(*
	Function for motion control of single axis.
	Provides an interface to PLC Open motion control blocks.
	Controls linking of limit switches from slave to master axes.
*)
FUNCTION_BLOCK FB_AxisDrive
VAR_INPUT
END_VAR
VAR_IN_OUT
	AxisController		:	ST_AxisControl;
END_VAR
VAR_OUTPUT
END_VAR
VAR
	eCommandLatched		:	eMcCommand;		//Internally latched command signal, new commands cannot be issued until existing commands have completed.
	doneLatch	:	SR;						//Used to set done signal in AxisController DUT
	bDone		:	BOOL;					//Interal done flag which will be used for latching on an external done located in AxisController DUT
	iParam		:	INT:=1;					//index of NC parameters FBs, no 0 index on array so initialised to 1
	iIndex		:	UINT;					//index value used for limit coupling
	iMasterIndex		:	UINT;			//index value used for limit coupling
	
	//Boolean to store EnableFw and EnableBw of MCPower FB
	FwLimitsEnabled	:	BOOL;	
	BWLimitsEnabled	:	BOOL;
	
	mcDirection	:	MC_Direction;			//Direction control required in function blocks

(*
Motion Function blocks taken from the PLC OPEN standard as defined by PLC Open Standard
Function blocks commented out are yet to be added but the intention is to add these.
Those listed as //NOT IMPLEMENTED have come from the standard but Beckhoff do not support, 
these have been added just as a placeholder for future support.
*)
	//Not Implemented
	//MCReadDigitalInput		:	MC_ReadDigitalInput;			//NOT IMPLEMENTED		
	//MCReadDigitalOutput		:	MC_ReadDigitalOutput;			//NOT IMPLEMENTED	
	//MCWriteDigitalOutput		:	MC_WriteDigitalOutput;			//NOT IMPLEMENTED
	//MCReadActualTorque		:	MC_ReadActualTorque;			//NOT IMPLEMENTED	
	//MCReadAxisInfo			:	MC_ReadAxisInfo;				//NOT IMPLEMENTED	
	//MCReadMotionState			:	MC_ReadMotionState;				//NOT IMPLEMENTED
	//MCDigitalCamSwitch		:	MC_DigitalCamSwitch;			//NOT IMPLEMENTED
	//MCTorqueControl			:	MC_TorqueControl;				//NOT IMPLEMENTED		
	//MCPositionProfile			:	MC_PositionProfile;				//NOT IMPLEMENTED		
	//MCVelocityProfile			:	MC_VelocityProfile;				//NOT IMPLEMENTED		
	//MCAccelerationProfile		:	MC_AccelerationProfile;			//NOT IMPLEMENTED
	
	
	(* Administrative Function Blocks *)                                                                     
	MCReset						:	MC_Reset;											
	MCPower						:	MC_Power;										
	//MCReadStatus				:	MC_ReadStatus;					//Same as Axis.ReadStatus();						
	//MCReadAxisError			:	MC_ReadAxisError;									
	MCReadParameter				:	MC_ReadParameter;														
	MCWriteParameter			:	MC_WriteParameter;										
	MCWriteBoolParameter		:	MC_WriteBoolParameter;								
		
	//MCReadActualPosition		:	MC_ReadActualPosition;								
	//MCReadActualVelocity		:	MC_ReadActualVelocity;								
		
	MCSetPosition				:	MC_SetPosition;										
	//MCSetOverride				:	MC_SetOverride;										
	//MCTouchProbe				:	MC_TouchProbe;										
		
	//MCAbortTrigger			:	MC_AbortTrigger;									
	//MCAbortSuperposition		:	MC_AbortSuperposition;			//Listed as HaltSuperimposed in PLC Open standard	
	//MCCamTableSelect			:	MC_CamTableSelect;									
	
	(* Motion Function Blocks *)
	//MCHome					:	MC_Home;											
	MCJog						:	MC_Jog;												
	MCStop						:	MC_Stop;											
	//MCHalt					:	MC_Halt;											
	MCMoveAbsolute				:	MC_MoveAbsolute;									
	MCMoveRelative				:	MC_MoveRelative;									
	//MCMoveAdditive			:	MC_MoveAdditive;									
	//MCMoveSuperimposed		:	MC_MoveSuperimposed;								
	MCMoveVelocity				:	MC_MoveVelocity;									
	//MCMoveContinuousAbsolute	:	MC_MoveContinuousAbsolute;						
	//MCMoveContinuousRelative	:	MC_MoveContinuousRelative;						
	//MCMoveModulo				:	MC_MoveModulo;										
	
	(* Synchronised Motion Function Blocks *)		
	MCGearIn					:	MC_GearIn;											
	//MCGearInDyn				:	MC_GearInDyn;										
	MCGearInMultiMaster			:	MC_GearInMultiMaster;								
	MCGearOut					:	MC_GearOut;												                                                                                    
	//MCHaltPhasing				:	MC_HaltPhasing;										
	//MCPhasingAbsolute			:	MC_PhasingAbsolute;									
	//MCPhasingRelative			:	MC_PhasingRelative;										                                                                                                                                                 
	//MCCamIn					:	MC_CamIn;											
	//MCCamOut					:	MC_CamOut;											
	//MCCamScaling				:	MC_CamScaling;										                                                      
	//MCCamAdd					:	MC_CamAdd;											
	//MCCamExchange				:	MC_CamExchange;										
	//MCCamInV2					:	MC_CamIn_V2;		//REQUIRED FOR MULTICAMMING 	
	//MCCamRemove				:	MC_CamRemove;										
	//MCCamScalingV2			:	MC_CamScaling_V2;									

	(* Advanced Homing Steps and Finishing Moves *)
	MCFinishHoming			:	MC_FinishHoming;
	//MCHomeDirect			:	MC_HomeDirect;
	//MCAbortHoming			:	MC_AbortHoming;
	MCStepAbsoluteSwitch	:	MC_StepAbsoluteSwitch;
	//MCStepBlock			:	MC_StepBlock;
	//MCStepBlockLagBased	:	MC_StepBlockLagBased;
	//MCStepLimitSwitch		:	MC_StepLimitSwitch;
	//MCStepReferencePulse	:	MC_StepReferencePulse;
	
	
	(* Additional variable structures required for Advanced Homing *)
	//MCSignalRef			:	MC_Ref_Signal_Ref;
	StOptions				:	ST_Home_Options;
	StOptions2				:	ST_Home_Options2;
	StOptions3				:	ST_Home_Options3;
	StOptions4				:	ST_Home_Options4;
	MCHomingParameter		:	MC_HomingParameter;		//Must be passed between homing steps.		
							
		
END_VAR

AxisController.Axis.ReadStatus();
AxisController.fActPosition:= AxisController.Axis.NcToPlc.ActPos;
AxisController.fActVelocity:= AxisController.Axis.NcToPlc.ActVelo;
AxisController.bNegativeDirection:= AxisController.Axis.status.NegativeDirection;
AxisController.bPositiveDirection:= AxisController.Axis.Status.PositiveDirection;
AxisController.bCalibrated:= AxisController.Axis.Status.Homed;

//////////////////////////////////////////////////////////////////////
//     _   __  _____ ____    ____ _____  _  _____ _____ ____  		//
//    / \  \ \/ |_ _/ ___|  / ___|_   _|/ \|_   _| ____/ ___| 		//
//   / _ \  \  / | |\___ \  \___ \ | | / _ \ | | |  _| \___ \ 		//
//  / ___ \ /  \ | | ___) |  ___) || |/ ___ \| | | |___ ___) |		//
// /_/   \_/_/\_|___|____/  |____/ |_/_/   \_|_| |_____|____/ 		//
// 																	//
//////////////////////////////////////////////////////////////////////
                                                            
//Numerical representation for axis states - may use later for buffering functions.
IF AxisController.AXIS.Status.Disabled THEN
	AxisController.iAxisState:=		100;
ELSIF AxisController.AXIS.Status.StandStill THEN
	AxisController.iAxisState:=		200;
ELSIF AxisController.AXIS.Status.Homing	THEN
	AxisController.iAxisState:= 	300;
ELSIF AxisController.AXIS.Status.DiscreteMotion	THEN
	AxisController.iAxisState:=		400;
ELSIF AxisController.AXIS.Status.SynchronizedMotion	THEN
	AxisController.iAxisState:=		500;
ELSIF AxisController.AXIS.Status.ContinuousMotion	THEN
	AxisController.iAxisState:=		600;
ELSIF AxisController.AXIS.Status.Stopping	THEN
	AxisController.iAxisState:= 	700;	
ELSIF AxisController.AXIS.Status.Error THEN
	AxisController.iAxisState:=		999;	
ELSE
	AxisController.iAxisState:=		0;
END_IF

//////////////////////////////////////////////////////////////////////////////////////////
//  _     ___ __  __ ___ _____   ______        _____ _____ ____ _   _ _____ ____  		//
// | |   |_ _|  \/  |_ _|_   _| / ___\ \      / |_ _|_   _/ ___| | | | ____/ ___| 		//
// | |    | || |\/| || |  | |   \___ \\ \ /\ / / | |  | || |   | |_| |  _| \___ \ 		//
// | |___ | || |  | || |  | |    ___) |\ V  V /  | |  | || |___|  _  | |___ ___) |		//
// |_____|___|_|  |_|___| |_|   |____/  \_/\_/  |___| |_| \____|_| |_|_____|____/		//
//																						//
//////////////////////////////////////////////////////////////////////////////////////////

//Initialise Foward and Backward limits to the hardware limit switches for this axis
FwLimitsEnabled :=Limits.FwLimit[GVL.iAxis];
BwLimitsEnabled :=Limits.BwLimit[GVL.iAxis];

(*
Cycle through Limits.coupledFwLimit and Limits.coupledBwLimit.
Looking to see if any axes have the current axis (GVL.iAxis) listed as a master.
If this axis is listed as a master, check the hardware limits of that slave.
Gear ratio determines whether we are looking for a Forward or a Backward limit on the slave axis. 
If the limit switch is disabled, disable motion for this axis.
*)
FOR iIndex:=1 TO GVL.axisNumMax DO
	FOR iMasterIndex:=1 TO 5 DO
		//If listed as a master
		IF Limits.coupledFwLimit[iIndex][iMasterIndex].iMasterAxis = GVL.iAxis THEN
			//If forward limit linked to forward of slave, check forward limit of slave
			IF Limits.coupledFwLimit[iIndex][iMasterIndex].eLimitType=eLimitCoupling.FwSw AND NOT Limits.FwLimit[iIndex] THEN
				FwLimitsEnabled:=FALSE;
			END_IF
			//If forward limit linked to backwardof slave, check forward limit of slave
			IF Limits.coupledFwLimit[iIndex][iMasterIndex].eLimitType=eLimitCoupling.BwSw AND NOT Limits.BwLimit[iIndex] THEN
				FwLimitsEnabled:=FALSE;
			END_IF
			//If backward limit linked to forward of slave, check forward limit of slave
			IF Limits.coupledBwLimit[iIndex][iMasterIndex].eLimitType=eLimitCoupling.FwSw AND NOT Limits.FwLimit[iIndex] THEN
				BwLimitsEnabled:=FALSE;
			END_IF
			//If backward limit linked to backward of slave, check backward limit of slave
			IF Limits.coupledBwLimit[iIndex][iMasterIndex].eLimitType=eLimitCoupling.BwSw AND NOT Limits.BwLimit[iIndex] THEN
				BwLimitsEnabled:=FALSE;
			END_IF
		END_IF
	END_FOR
END_FOR

AxisController.bFwEnabled:=FwLimitsEnabled;		//Feedback to ST_AxisControl that forward positioning is available
AxisController.bBwEnabled:=BwLimitsEnabled;		//Feedback to ST_AxisControl that backward positioning is available

//////////////////////////////////////////////////////////
//  ____   _____        _______ ____    _   _ ____  	//
// |  _ \ / _ \ \      / | ____|  _ \  | | | |  _ \ 	//
// | |_) | | | \ \ /\ / /|  _| | |_) | | | | | |_) |	//
// |  __/| |_| |\ V  V / | |___|  _ <  | |_| |  __/ 	//
// |_|    \___/  \_/\_/  |_____|_| \_\  \___/|_|   		//
//														//
//////////////////////////////////////////////////////////
(*
Power up the axis.
Externally fed variables are bEnabled and fOverride, limits all controlled internally.
*)                                           
MCPower(
	Axis:=AxisController.Axis,
	Enable:=AxisController.bEnable,
	Enable_Positive:=FwLimitsEnabled,
	Enable_Negative:=BwLimitsEnabled,
	Override:=AxisController.fOverride,
	Status=>,
	Busy=>, 
	Active=>AxisController.bAxisReady,	//Maybe want a bPowered or bEnabled flag instead?
	Error=>,
	ErrorID=>
);

//////////////////////////////////////////////////////////////////////////////////////////////////////////
//  ____  _____    _    ____    ____   _    ____     _    __  __ _____ _____ _____ ____  ____  			//
// |  _ \| ____|  / \  |  _ \  |  _ \ / \  |  _ \   / \  |  \/  | ____|_   _| ____|  _ \/ ___| 			//
// | |_) |  _|   / _ \ | | | | | |_) / _ \ | |_) | / _ \ | |\/| |  _|   | | |  _| | |_) \___ \ 			//
// |  _ <| |___ / ___ \| |_| | |  __/ ___ \|  _ < / ___ \| |  | | |___  | | | |___|  _ < ___) |			//
// |_| \_|_____/_/   \_|____/  |_| /_/   \_|_| \_/_/   \_|_|  |_|_____| |_| |_____|_| \_|____/ 			//
//                                                                                           			//
//////////////////////////////////////////////////////////////////////////////////////////////////////////
(*
Check NC parameters available from MCReadParameter FB (17 in total)
See eRWParameter DUT for complete list or PLC OPEN documentation
To call all 17 from a single functionblock instance only 1 can be checked per cycle so there will be at minimum a 34 cycle delay checking each parameter
The MCReadParameter does also cover the functionality of MCReadBoolParameter so these booleans are separately converted from the MCReadParameter call
*)
MCReadParameter(Axis:=AxisController.AXIS,ParameterNumber:=iParam);
IF MCReadParameter.Valid THEN
	MCReadParameter.Enable:=FALSE;
	AxisController.fParameters[iParam]:=MCReadParameter.Value;
	iParam:= iParam+1;
	IF iParam>17 THEN
		iParam:=1;
	END_IF
ELSE
	MCReadParameter.Enable:=TRUE;
END_IF

//Convert LREALS to BOOLS


IF AxisController.fParameters[eRWParameter.EnableLimitPos]=1 THEN
	AxisController.bSoftLimPosEn:=TRUE;
ELSE
	AxisController.bSoftLimPosEn:=FALSE;
END_IF
IF AxisController.fParameters[eRWParameter.EnableLimitNeg]=1 THEN
	AxisController.bSoftLimNegEn:=TRUE;
ELSE
	AxisController.bSoftLimNegEn:=FALSE;
END_IF
IF AxisController.fParameters[eRWParameter.EnablePosLagMonitoring]=1 THEN
	AxisController.bPosLagEn:=TRUE;
ELSE
	AxisController.bPosLagEn:=FALSE;
END_IF

//////////////////////////////////////////////////////////////////////////////////////////////////////////
//  __  __  ____   _____ _   _ _   _  ____ _____ ___ ___  _   _    ____    _    _     _     ____  		//
// |  \/  |/ ___| |  ___| | | | \ | |/ ___|_   _|_ _/ _ \| \ | |  / ___|  / \  | |   | |   / ___| 		//
// | |\/| | |     | |_  | | | |  \| | |     | |  | | | | |  \| | | |     / _ \ | |   | |   \___ \ 		//
// | |  | | |___  |  _| | |_| | |\  | |___  | |  | | |_| | |\  | | |___ / ___ \| |___| |___ ___) |		//
// |_|  |_|\____| |_|    \___/|_| \_|\____| |_| |___\___/|_| \_|  \____/_/   \_|_____|_____|____/ 		//
//                                         																//                                                      
//////////////////////////////////////////////////////////////////////////////////////////////////////////
(*
Call MC Function Blocks and clear execute signals
Any MC function blocks added to the state machine must be called here with the given format.
Some FBs have slightly differing structures so these should aim to conform to the existing structure
Function blocks will hold done and error signals for 1 cycle with no execute held
*)
MCReadParameter(Axis:=AxisController.Axis);	//Reading in motion parameters, using one functionblock for all params means need to disable

MCReset(Axis:=AxisController.Axis);
MCReset.Execute:=FALSE;

MCWriteParameter(Axis:=AxisController.Axis);
MCWriteParameter.Execute:=FALSE;

MCWriteBoolParameter(Axis:=AxisController.Axis);
MCWriteBoolParameter.Execute:=FALSE;

MCSetPosition(Axis:=AxisController.Axis);
MCSetPosition.Execute:=FALSE;

MCMoveAbsolute(Axis:=AxisController.Axis);
MCMoveAbsolute.Execute:=FALSE;

MCMoveRelative(Axis:=AxisController.Axis);
MCMoveRelative.Execute:=FALSE;

MCGearIn(Slave:=AxisController.Axis, Master:=GVL.axes[AxisController.masterAxis].Axis);
MCGearIn.Execute:=FALSE;

MCGearInMultiMaster(Master1:=GVL.axes[AxisController.masterAxes[1].i].Axis,Master2:=GVL.axes[AxisController.masterAxes[2].i].Axis,Master3:=GVL.axes[AxisController.masterAxes[3].i].Axis,Master4:=GVL.axes[AxisController.masterAxes[4].i].Axis,Slave:=AxisController.Axis);
MCGearInMultiMaster.Enable:=FALSE;	//NOT EXECUTE AS FB ALLOWS CONTINUAL UPDATING OF RATIOS WHILST ENABLED

MCGearOut(Slave:=AxisController.Axis);
MCGearOut.Execute:=FALSE;

MCJog(Axis:=AxisController.Axis);
MCJog.JogBackwards:=FALSE;
MCJog.JogForward:=FALSE;

MCStepAbsoluteSwitch(Axis:=AxisController.Axis,Parameter:=MCHomingParameter);
MCStepAbsoluteSwitch.Execute:=FALSE;


MCFinishHoming(Axis:=AxisController.Axis,Parameter:=MCHomingParameter);
MCFinishHoming.Execute:=FALSE;

MCMoveVelocity(Axis:=AxisController.Axis);
MCMoveVelocity.Execute:=FALSE;

MCStop(Axis:=AxisController.Axis);
MCStop.Execute:=FALSE;

//////////////////////////////////////////////////////////////////////////////////////////////////////////////////////////////////////////////
//   ____ ___  __  __ __  __    _    _   _ ____     ____    _    ____  _____   ____ _____  _  _____ _____ __  __ _____ _   _ _____ ____ 	// 
//  / ___/ _ \|  \/  |  \/  |  / \  | \ | |  _ \   / ___|  / \  / ___|| ____| / ___|_   _|/ \|_   _| ____|  \/  | ____| \ | |_   _/ ___| 	//
// | |  | | | | |\/| | |\/| | / _ \ |  \| | | | | | |     / _ \ \___ \|  _|   \___ \ | | / _ \ | | |  _| | |\/| |  _| |  \| | | | \___ \ 	//
// | |__| |_| | |  | | |  | |/ ___ \| |\  | |_| | | |___ / ___ \ ___) | |___   ___) || |/ ___ \| | | |___| |  | | |___| |\  | | |  ___) |	//
//  \____\___/|_|  |_|_|  |_/_/   \_|_| \_|____/   \____/_/   \_|____/|_____| |____/ |_/_/   \_|_| |_____|_|  |_|_____|_| \_| |_| |____/	//
//																																			//
//////////////////////////////////////////////////////////////////////////////////////////////////////////////////////////////////////////////

(*
Internal statemachine to handle motion control flow and logic.
Functions are NOT called in this statemachine, these just update values given to the state machine. This was the method recommended by Beckhoff
The following basic wrapper should be used for adding new function blocks. Any that do not conform to this should be modified to conform
Notably some FBs have no .Done but do have .Active
	
	mcFunctionBlock.Execute		:=AxisController.bExecute;
	mcFunctionBlock.misc1..n	:=AxisController.misc1..n;
	
	bDone:=mcFunctionBlock.Done;
	AxisController.bBusy:= mcFunctionBlock.Busy;
	
	If mcFunctionBlock.Error THEN
		AxisController.bError:=TRUE;
		AxisController.iErrorID:= mcFunctionBlock.ErrorID;
	END_IF
	IF NOT mcFunctionBlock.Busy THEN
		eCommandLatched:=eMcCommand.Idle;
	END_IF
	
Function block specific parameters should be added to the ST_AxisControl if not already listed
eCommandLatched is currently being used to hold control flow logic so that users cannot send new commands until previous ones have complete.
This will definitely need to be modified to allow buffering in the future and to allow stop/halt commands 
but I haven't looked in to the best way to do this yet.	

It may be that it doesn't matter if it is latched at all as we can rely on waiting for the done signal before sending subsequent commands if it really matters
*)
//If we're not doing anything or have just done something we no longer latch on the given command
eCommandLatched:=AxisController.eCommand;

CASE eCommandLatched OF
	
	eMcCommand.Idle:
		AxisController.bBusy	:=FALSE;
		AxisController.bExecute	:=FALSE;
///////////////////////////////////////////////////////////////////////////////////////////////////////////////////////////////	
	eMcCommand.Reset:
		AxisController.bError	:=FALSE;
		MCReset.Execute:=AxisController.bReset;
		
		bDone:=McReset.Done;
		AxisController.bBusy:=MCReset.Busy;
		IF MCReset.Error THEN
			AxisController.bError:=TRUE;
			AxisController.iErrorID:=MCReset.ErrorID;	
		END_IF
		IF NOT MCReset.Busy THEN
			eCommandLatched:=eMcCommand.Idle;
			AxisController.bReset:=FALSE;
		END_IF
///////////////////////////////////////////////////////////////////////////////////////////////////////////////////////////////
	eMcCommand.WriteParameter:		
		MCWriteParameter.Execute:=AxisController.bExecute;
		MCWriteParameter.ParameterNumber:=AxisController.iParameterIndex;
		MCWriteParameter.Value:=AxisController.fParameterValue;
		
		bDone:=MCWriteParameter.Done;
		AxisController.bBusy:= MCWriteParameter.Busy;
		
		IF MCWriteParameter.Error THEN
			AxisController.bError:=TRUE;
			AxisController.iErrorID:=MCWriteParameter.ErrorID;	
		END_IF	
		IF NOT MCWriteParameter.Busy THEN
			eCommandLatched:=eMcCommand.Idle;
		END_IF			
///////////////////////////////////////////////////////////////////////////////////////////////////////////////////////////////
	eMcCommand.WriteBoolParameter:	
		MCWriteBoolParameter.Execute:=AxisController.bExecute;
		MCWriteBoolParameter.ParameterNumber:=AxisController.iParameterIndex;
		MCWriteBoolParameter.Value:=AxisController.bInput;
		
		bDone:=MCWriteBoolParameter.Done;
		AxisController.bBusy:=MCWriteBoolParameter.Busy;
		
		IF MCWriteBoolParameter.Error THEN
			AxisController.bError:= TRUE;
			AxisController.iErrorID:=MCWriteBoolParameter.ErrorID;
		END_IF			
		IF NOT MCWriteBoolParameter.Busy THEN
			eCommandLatched:=eMcCommand.Idle;
		END_IF	
///////////////////////////////////////////////////////////////////////////////////////////////////////////////////////////////
	eMcCommand.SetPosition:	
		MCSetPosition.Execute:=AxisController.bExecute;
		MCSetPosition.Position:=AxisController.fPosition;
		
		AxisController.bBusy:=MCSetPosition.Busy;
		bDone:=MCSetPosition.Done;
		
		IF MCSetPosition.Error THEN
			AxisController.bError:=TRUE;
			AxisController.iErrorID:= MCSetPosition.ErrorID;
		END_IF
		IF NOT MCSetPosition.Busy THEN
			eCommandLatched:=eMcCommand.Idle;
		END_IF
///////////////////////////////////////////////////////////////////////////////////////////////////////////////////////////////
	eMcCommand.MoveAbsolute:	
		MCMoveAbsolute.Execute:=AxisController.bExecute;
		MCMoveAbsolute.Position:=AxisController.fPosition;
		MCMoveAbsolute.Velocity:=AxisController.fVelocity;
		MCMoveAbsolute.Acceleration:=AxisController.fAcceleration;
		MCMoveAbsolute.Deceleration:=AxisController.fDeceleration;
		MCMoveAbsolute.Jerk:=0;
		//MCMoveAbsolute.BufferMode:=MC_BufferMode.MC_Buffered;
		
		bDone:=MCMoveAbsolute.Done;
		AxisController.bBusy:=MCMoveAbsolute.Busy;
		
		IF MCMoveAbsolute.Error THEN
			AxisController.bError:=TRUE;
			AxisController.iErrorID:=MCMoveAbsolute.ErrorID;
		END_IF
		IF NOT MCMoveAbsolute.Busy THEN
			eCommandLatched:=eMcCommand.Idle;
		END_IF
///////////////////////////////////////////////////////////////////////////////////////////////////////////////////////////////
	eMcCommand.MoveRelative:		
		MCMoveRelative.Execute:=AxisController.bExecute;
		MCMoveRelative.Distance:=AxisController.fDistance;
		MCMoveRelative.Velocity:=AxisController.fVelocity;
		MCMoveRelative.Acceleration:=AxisController.fAcceleration;
		MCMoveRelative.Deceleration:=AxisController.fDeceleration;
		MCMoveRelative.Jerk:=0;
		//MCMoveRelative.BufferMode:=MC_BufferMode.MC_Buffered;
		
		bDone:=MCMoveRelative.Done;
		AxisController.bBusy:=MCMoveRelative.Busy;
		
		IF MCMoveRelative.Error THEN
			AxisController.bError:=TRUE;
			AxisController.iErrorID:=MCMoveRelative.ErrorID;
		END_IF
		IF NOT MCMoveRelative.Busy THEN
			eCommandLatched:=eMcCommand.Idle;
		END_IF		
///////////////////////////////////////////////////////////////////////////////////////////////////////////////////////////////
	eMcCommand.GearIn:
		//Dependent on +ve or -ve gear ratio determines whether to link Fw to Fw and Bw to Bw or Fw to Bw and Bw to Fw
		IF AxisController.fGearRatioNum>0 THEN
			Limits.coupledFwLimit[GVL.iAxis][1].eLimitType:=eLimitCoupling.FwSw;		
			Limits.coupledBwLimit[GVL.iAxis][1].eLimitType:=eLimitCoupling.BwSw;				
		END_IF
		IF AxisController.fGearRatioNum<0 THEN
			Limits.coupledFwLimit[GVL.iAxis][1].eLimitType:=eLimitCoupling.BwSw;
			Limits.coupledBwLimit[GVL.iAxis][1].eLimitType:=eLimitCoupling.FwSw;		
		END_IF
		Limits.coupledFwLimit[GVL.iAxis][1].iMasterAxis:=AxisController.masterAxis;
		Limits.coupledBwLimit[GVL.iAxis][1].iMasterAxis:=AxisController.masterAxis;
		
		MCGearIn.Execute:=AxisController.bExecute;
		MCGearIn.RatioNumerator:=AxisController.fGearRatioNum;
		MCGearIn.RatioDenominator:=AxisController.iGearRatioDen;
		
		bDone:=McGearIn.InGear;
		AxisController.bBusy:=MCGearIn.Busy;
		
		IF MCGearIn.Error THEN
			AxisController.bError:=TRUE;
			AxisController.iErrorID:=MCGearIn.ErrorID;
		END_IF		
		IF NOT MCGearIn.Busy THEN
			eCommandLatched:=eMcCommand.Idle;
		END_IF
///////////////////////////////////////////////////////////////////////////////////////////////////////////////////////////////
	eMcCommand.GearInMultiMaster:		
		//Set up limits
		FOR iMasterIndex:=1 TO GVL.axisCoupleMax DO
			IF AxisController.masterAxes[iMasterIndex].ratio>0 THEN
				Limits.coupledFwLimit[GVL.iAxis][iMasterIndex+1].eLimitType:=eLimitCoupling.FwSw;				
				Limits.coupledBwLimit[GVL.iAxis][iMasterIndex+1].eLimitType:=eLimitCoupling.BwSw;				
			END_IF
			IF AxisController.masterAxes[iMasterIndex].ratio<0 THEN
				Limits.coupledFwLimit[GVL.iAxis][iMasterIndex+1].eLimitType:=eLimitCoupling.BwSw;
				Limits.coupledBwLimit[GVL.iAxis][iMasterIndex+1].eLimitType:=eLimitCoupling.FwSw;
			END_IF
			Limits.coupledFwLimit[GVL.iAxis][iMasterIndex+1].iMasterAxis:=AxisController.masterAxes[iMasterIndex].i;
			Limits.coupledBwLimit[GVL.iAxis][iMasterIndex+1].iMasterAxis:=AxisController.masterAxes[iMasterIndex].i;
		END_FOR
		

		
		(*	Issue with this MC block (other than everything...) is that it doesn't conform to the standard and use an execute signal. The execute
			signal in any other block determines that when it is high one of either error,done,busy must be on. That is not the case with this block
			what happens is it triggers, doesn't register a busy and so immediately clears as done. If has been modified to conform.
		*)
		MCGearInMultiMaster.Enable:=AxisController.bExecute;
		MCGearInMultiMaster.GearRatio1:=AxisController.masterAxes[1].ratio;
		MCGearInMultiMaster.GearRatio2:=AxisController.masterAxes[2].ratio;
		MCGearInMultiMaster.GearRatio3:=AxisController.masterAxes[3].ratio;
		MCGearInMultiMaster.GearRatio4:=AxisController.masterAxes[4].ratio;
		
		AxisController.bBusy:=MCGearInMultiMaster.Busy;
		IF MCGearInMultiMaster.Enable THEN
			AxisController.bBusy:=TRUE;	//busy does not go immediately high when enable high 
			bDone:=FALSE;
		END_IF

		bDone:=MCGearInMultiMaster.InGear;	
		IF MCGearInMultiMaster.Error THEN
			AxisController.bError:=TRUE;
			AxisController.iErrorID:=MCGearInMultiMaster.ErrorID;
		END_IF
		IF NOT MCGearInMultiMaster.Busy THEN
			eCommandLatched:=eMcCommand.Idle;
		END_IF
///////////////////////////////////////////////////////////////////////////////////////////////////////////////////////////////
	eMcCommand.GearOut:		
		//Gearout - remove all masters from slave
		FOR iMasterIndex:=1 TO 5 DO
				Limits.coupledFwLimit[GVL.iAxis][iMasterIndex].eLimitType:=eLimitCoupling.None;
				Limits.coupledBwLimit[GVL.iAxis][iMasterIndex].eLimitType:=eLimitCoupling.None;
		END_FOR		
	
		MCGearOut.Execute:=AxisController.bExecute;
		
		AxisController.bBusy:=MCGearOut.Busy;
		bDone:=MCGearOut.Done;
		IF MCGearOut.Error THEN
			AxisController.bError:=TRUE;
			AxisController.iErrorID:=MCGearOut.ErrorID;
		END_IF
		IF NOT MCGearOut.Busy THEN
			eCommandLatched:=eMcCommand.Idle;
		END_IF
	///////////////////////////////////////////////////////////////////////////////////////////////////////////////////////////////			
	eMcCommand.Jog:
		MCJog.JogForward:=AxisController.bJogForward;
		MCJog.JogBackwards:=AxisController.bJogBackward;
		
		bDone:=MCJog.Done;
		
		IF MCJog.Error THEN
			AxisController.bError:=TRUE;
			AxisController.iErrorID:=MCJog.ErrorID;
		END_IF
		IF NOT MCJog.Busy THEN
			eCommandLatched:=eMcCommand.Idle;
		END_IF
	///////////////////////////////////////////////////////////////////////////////////////////////////////////////////////////////	
	eMcCommand.HomeStepAbsoluteSwitch:
		//Issue: If execute not held high the function will not reverse on its own to find the abs switch when hitting a limit
		//You have to reissue the command. I want to try and keep bExecute high
		IF (NOT Limits.FwLimit[GVL.iAxis]) OR (NOT Limits.BwLimit[GVL.iAxis]) THEN
			MCStepAbsoluteSwitch.Execute:=TRUE;
		ELSE	
			MCStepAbsoluteSwitch.Execute:=AxisController.bExecute;
		END_IF
	
		MCStepAbsoluteSwitch.Direction:= AxisController.mcHomeDirection;
		MCStepAbsoluteSwitch.SwitchMode:=AxisController.mcSwitchMode;
		MCStepAbsoluteSwitch.ReferenceSignal:=AxisController.mcSignalRef;
		MCStepAbsoluteSwitch.Velocity:=AxisController.fHomeVelocity;
		MCStepAbsoluteSwitch.Acceleration:=0;
		MCStepAbsoluteSwitch.Deceleration:=0;
		MCStepAbsoluteSwitch.Jerk:=0;
		MCStepAbsoluteSwitch.TorqueLimit:=AxisController.fHomeTorque;
		MCStepAbsoluteSwitch.SetPosition:=AxisController.fHomePosition;
		MCStepAbsoluteSwitch.TimeLimit:=AxisController.tHomeTimeLimit;
		MCStepAbsoluteSwitch.DistanceLimit:=AxisController.fHomeDistanceLimit;
		MCStepAbsoluteSwitch.PositiveLimitSwitch:= NOT Limits.FwLimit[GVL.iAxis];	//Step FB has R_TRIG behaviour but limits set as Normally Closed so logic is inverted
		MCStepAbsoluteSwitch.NegativeLimitSwitch:= NOT Limits.BwLimit[GVL.iAxis];	//Step FB has R_TRIG behaviour but limits set as Normally Closed so logic is inverted
		MCStepAbsoluteSwitch.BufferMode:=AxisController.buffer;
		StOptions4.DisableDriveAccess:=TRUE;		//Testing required with hardware. This step may be redundant.
		MCStepAbsoluteSwitch.Options:=StOptions4;
		
		bDone:=MCStepAbsoluteSwitch.Done;
		AxisController.bBusy:=MCStepAbsoluteSwitch.Busy;
		
		IF MCStepAbsoluteSwitch.Error THEN
			AxisController.bError:=TRUE;
			AxisController.iErrorID:=MCStepAbsoluteSwitch.ErrorID;
		END_IF
		IF NOT MCStepAbsoluteSwitch.Busy THEN
			eCommandLatched:=eMcCommand.Idle;
		END_IF
	///////////////////////////////////////////////////////////////////////////////////////////////////////////////////////////////	
	eMcCommand.HomeFinish:
		MCFinishHoming.Execute:=AxisController.bExecute;
		MCFinishHoming.Distance:=AxisController.fHomeDistance;
		MCFinishHoming.Velocity:=AxisController.fHomeVelocity;
		
		StOptions2.DisableDriveAccess:=TRUE;	//Testing required with hardware. This step may be redundant.
		MCFinishHoming.Options:=StOptions2;
		
		bDone:=MCFinishHoming.Done;
		AxisController.bBusy:=MCFinishHoming.Busy;
		
		IF MCFinishHoming.Error THEN
			AxisController.bError:=TRUE;
			AxisController.iErrorID:=MCFinishHoming.ErrorID;
		END_IF
		IF NOT MCFinishHoming.Busy THEN
			eCommandLAtched:=eMcCommand.Idle;
		END_IF
	///////////////////////////////////////////////////////////////////////////////////////////////////////////////////////////////	
	eMcCommand.MoveVelocity:
		MCMoveVelocity.Execute:=AxisController.bExecute;
		MCMoveVelocity.Acceleration:=AxisController.fAcceleration;
		MCMoveVelocity.Deceleration:=AxisController.fDeceleration;
		
		//Simple logic to allow negative velocity inputs rather than having to set the direction object
		IF AxisController.fVelocity>= 0 THEN
			MCMoveVelocity.Velocity:=AxisController.fVelocity;
			MCMoveVelocity.Direction:= MC_Positive_Direction;
		ELSE
			MCMoveVelocity.Velocity:=ABS(AxisController.fVelocity);
			MCMoveVelocity.Direction:= MC_Negative_Direction;
		END_IF
		
		bDone:=MCMoveVelocity.InVelocity;
		AxisController.bBusy:=MCMoveVelocity.Busy;
		
		IF MCMoveVelocity.Error THEN
			AxisController.bError:=TRUE;
			AxisController.iErrorID:=MCMoveVelocity.ErrorID;
		END_IF
		IF NOT MCMoveVelocity.Busy THEN
			eCommandLatched:=eMcCommand.Idle;
		END_IF
	///////////////////////////////////////////////////////////////////////////////////////////////////////////////////////////////	
	eMcCommand.Stop:
		McStop.Execute:=AxisController.bExecute;
		McStop.Deceleration:=AxisController.fDeceleration;
		McStop.Jerk:=0;
		
		bDone:=McStop.Done;
		AxisController.bBusy:=McStop.Busy;
		
		IF MCStop.Error THEN
			AxisController.bError:= TRUE;
			AxisController.iErrorID:=MCStop.ErrorId;
		END_IF
		IF	NOT MCStop.Busy THEN
			eCommandLatched:=eMcCommand.Idle;
		END_IF

		
END_CASE

////////////////////////////////////////// 
//  _____ _        _    ____ ____  		//
// |  ___| |      / \  / ___/ ___| 		//
// | |_  | |     / _ \| |  _\___ \ 		//
// |  _| | |___ / ___ | |_| |___) |		//
// |_|   |_____/_/   \_\____|____/ 		//
//                                		//
//////////////////////////////////////////
AxisController.bMoving:=AxisController.Axis.Status.Moving;	
AxisController.bExecute:=FALSE;

(*
As we never hold Execute high, the done signal from each function block will only stay on for 1 cycle tick
The following logic just uses an SR latch to hold this done signal TRUE until it is cleared either by an error or the axis going busy

Errors are always latched as they are only ever set by a FB error and cleared by a reset command
*)
doneLatch(SET1:=bDone,RESET:=(AxisController.bBusy OR AxisController.bError));
AxisController.bDone:=doneLatch.Q1;

END_FUNCTION_BLOCK

(* stored: Version 1.1.0.1, ProductVersion 3.1.4022.12
   POU FB_AxisDrive: Id {aef7aef0-3971-449b-83a3-6f8c4c2f7d04}, SpecialFunc None *)
